FUNCTION_BLOCK FB_CommandChangeStop EXTENDS FB_CommandChange IMPLEMENTS ITF_CommandChange
VAR

END_VAR

(*			
	RafalOS
	Rafał Osajda		03.11.2025		TC 4024.66
	Test czy można zmienić stan lub tryb i zwraca czy można i uruchamia zmianę
*)
METHOD PUBLIC Execute : BOOL
VAR_INPUT
	iNumberOfCommand	: INT;
END_VAR
IF (THIS^.itfSaMController.GetState () = E_BaseMachineState.Resetting OR
	THIS^.itfSaMController.GetState () = E_BaseMachineState.Idle OR
	THIS^.itfSaMController.GetState () = E_BaseMachineState.Starting OR
	THIS^.itfSaMController.GetState () = E_BaseMachineState.Execute OR
	THIS^.itfSaMController.GetState () = E_BaseMachineState.Suspending OR
	THIS^.itfSaMController.GetState () = E_BaseMachineState.Suspended OR
	THIS^.itfSaMController.GetState () = E_BaseMachineState.Unsuspending OR
	THIS^.itfSaMController.GetState () = E_BaseMachineState.Holding OR
	THIS^.itfSaMController.GetState () = E_BaseMachineState.Held OR
	THIS^.itfSaMController.GetState () = E_BaseMachineState.Unholding OR
	THIS^.itfSaMController.GetState () = E_BaseMachineState.Completing OR
	THIS^.itfSaMController.GetState () = E_BaseMachineState.Complete) THEN		// sprawdzenie czy jesteśmy w dobrym stanie dla tego rozkazu
	IF (THIS^.itfSaMController.IsStateInModeEnabled (eStateIn := E_BaseMachineState.Stopping)) THEN	//test czy stan do którego chcemy przejśc jest właczony dla tego trybu
		THIS^.itfSaMController.ChangeStateTo (eStateIn := E_BaseMachineState.Stopping);
	ELSE
		THIS^.EventSetActive (iNumber := 5);	//stan docelowy jest wylaczony w tym trybie
	END_IF
ELSE
	THIS^.EventSetActive (iNumber := 4);	//ten rozkaz nie obsluguje tego stanu
END_IF
END_METHOD

METHOD FB_init : BOOL
VAR_INPUT
	bInitRetains : BOOL; // if TRUE, the retain variables are initialized (warm start / cold start)
	bInCopyCode : BOOL;  // if TRUE, the instance afterwards gets moved into the copy code (online change)
END_VAR
THIS^.SetText (eLocation := E_BaseLocation.pl, wsDescription := "Command change state - Stop");
THIS^.SetText (eLocation := E_BaseLocation.en, wsDescription := "Command change state - Stop");
THIS^.SetText (eLocation := E_BaseLocation.de, wsDescription := "Command change state - Stop");
THIS^.SetName (stName := THIS^.GetTexts ());
END_METHOD

END_FUNCTION_BLOCK

(* stored: Version 1.1.0.1
   POU FB_CommandChangeStop: Id {710e81c1-15d4-0880-22ef-20bc03f25b26}, SpecialFunc None
   Method Execute: Id {9e91b359-6ef7-0d97-2882-474326bf9133}
   Method FB_init: Id {9e12d0ec-1ea7-0a68-0f8e-851d274e0cb4} *)
